FUNCTION_BLOCK Q_LockUnlockMask (* Command Lock/UnlockMask( Part 6 - F.46 ) *)
  (* Standard: ISO 11783-6; Description: This message is available in VT Version 4 and later. This command is used by a Working Set to disallow or allow screen refreshes at the VT for the visible Data Mask or User-Layout Data Mask owned by the requesting Working Set. Return values iso_s16 - E_NO_ERR - OK - E_OVERFLOW - buffer overflow - E_NOACT - Command not possible in current state - E_NO_INSTANCE - No VT client available *)
  (* Version 1.0, 2022-07-08, franz *)
  (* Documentation:
  This message is available in VT Version 4 and later. This command is used by a Working Set to disallow or allow screen refreshes at the VT for the visible Data Mask or User-Layout Data Mask owned by the requesting Working Set.
   Return values
   iso_s16
    - E_NO_ERR - OK
   - E_OVERFLOW - buffer overflow
   - E_NOACT - Command not possible in current state
   - E_NO_INSTANCE - No VT client available
  *)
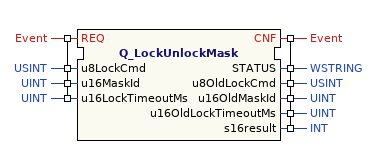
  EVENT_INPUT
    REQ WITH u8LockCmd, u16MaskId, u16LockTimeoutMs; (* Service Request *)
  END_EVENT
  EVENT_OUTPUT
    CNF WITH STATUS, s16result, u8OldLockCmd, u16OldMaskId, u16OldLockTimeoutMs; (* Confirmation of Requested Service *)
  END_EVENT
  VAR_INPUT
    u8LockCmd : USINT; (* 0 = Unlock, 1 = Lock data mask or user-layout data mask *)
    u16MaskId : UINT; (* Object ID of data mask or user layout data mask to lock or unlock *)
    u16LockTimeoutMs : UINT; (* Lock timeout in ms or zero for no timeout *)
  END_VAR
  VAR_OUTPUT
    STATUS : WSTRING; (* Service Status *)
    u8OldLockCmd : USINT; (* Old 0 = Unlock, 1 = Lock data mask or user-layout data mask *)
    u16OldMaskId : UINT; (* Old object ID of data mask or user layout data mask to lock or unlock *)
    u16OldLockTimeoutMs : UINT; (* Old lock timeout in ms or zero for no timeout *)
    s16result : INT; (* retval see description *)
  END_VAR
END_FUNCTION_BLOCK
